TYPE ST_AMI8000IOInfo :
STRUCT
	bAxisOperational 	: BOOL;
	bNotMoving			: BOOL;
	rActualPosition		: LREAL;
	rActualVelocity		: LREAL;
	rActualTorque		: LREAL;
	bAxisHomed			: BOOL;
	bAxisError			: BOOL;
	nErrorCode			: UDINT;
END_STRUCT
END_TYPE

(* stored: Version 1.1.0.1, ProductVersion 3.1.4024.12
   DUT ST_AMI8000IOInfo: Id {907b4956-497f-41ba-9b73-91c652065f98} *)
